TEXTLIST RunModeTypeTexList
  0 = '正常生产' | Chinese: '正常生产' | English: 'Normal Product'
  1 = '动态重复性' | Chinese: '动态重复性' | English: 'GRR'
  2 = '静态重复性' | Chinese: '静态重复性' | English: 'ARR'
   = ''
END_TEXTLIST

(* stored: Version 1.1.0.1, ProductVersion 3.1.4024.4
   TextList RunModeTypeTexList: Id {b8ce8886-2068-4cd8-a249-60604adb6f91} *)
